(* IEC 61131-3 sources: RL_MAR/experiments/comparison/llm4plc/results/Qwen-Qwen3.5-9B_20260506_150728/20260506_174552, 3 files *)

(* ---- generated_code_iteration_0.st ---- *)
START_ST
FUNCTION_BLOCK SolarPanelTracking
VAR
    PanelAngle : REAL; (* Output for adjusting the solar panel angle *)
    SunriseTime : TIME := T#6H; (* Set the time for sunrise (6:00 AM) *)
    SunsetTime : TIME := T#18H; (* Set the time for sunset (6:00 PM) *)
    NoonTime : TIME := T#12H; (* Set the time for solar noon (12:00 PM) *)
    MorningAngle : REAL := 30.0; (* Set the morning angle for panels *)
    NoonAngle : REAL := 60.0; (* Set the noon angle for panels *)
    EveningAngle : REAL := 30.0; (* Set the evening angle for panels *)
END_VAR
VAR_INPUT
    CurrentTime : TIME;
    SolarIntensity : REAL;
END_VAR
VAR
    state : INT; (* The FSM state variable (0=Night, 1=Morning, 2=Evening, 3=Override) *)
    prevState : INT; (* To track previous state if needed for complex logic *)
    currentAngle : REAL; (* Temporary variable to hold the calculated angle before assignment to output *)
END_VAR

(* Initialize state if this is the first execution or reset logic *)
IF NOT (CurrentTime > T#0) OR (CurrentTime < T#0) THEN
    state := 0;
ELSE
    (* Determine current state based on logic plan *)
    (* STATE 3: HIGH_INTENSITY_OVERRIDE_MODE takes precedence *)
    IF SolarIntensity >= 90.0 THEN
        state := 3;
    (* STATE 0: NIGHT_MODE *)
    ELSIF (CurrentTime < SunriseTime) OR (CurrentTime >= SunsetTime) THEN
        state := 0;
    (* STATE 1: MORNING_MODE *)
    ELSIF CurrentTime < NoonTime THEN
        state := 1;
    (* STATE 2: EVENING_MODE *)
    ELSE
        state := 2;
    END_IF;
END_IF;

(* Assign output based on the determined state *)
CASE state OF
    0: (* NIGHT_MODE *)
        currentAngle := 0.0;
    1: (* MORNING_MODE *)
        currentAngle := MorningAngle;
    2: (* EVENING_MODE *)
        currentAngle := EveningAngle;
    3: (* HIGH_INTENSITY_OVERRIDE_MODE *)
        currentAngle := NoonAngle;
    ELSE
        currentAngle := 0.0; (* Default safety value *)
END_CASE;

(* Update the output variable *)
PanelAngle := currentAngle;

END_FUNCTION_BLOCK
END_ST

(* ---- generated_code_iteration_1.st ---- *)
START_REASON
The validation feedback indicates a CODESYS compiler error: "应该用表达式代替 'T#0'" (Should use an expression instead of 'T#0').

In IEC 61131-3 Structured Text (ST), the literal `T#0` (representing 0 time) is often not accepted directly in boolean comparisons like `CurrentTime > T#0` or `CurrentTime < T#0` because the compiler expects a specific time expression or a comparison against a valid time value that resolves to a boolean context correctly in all dialects.

The standard and most robust way to check if a `TIME` variable is zero is to compare it against `T#0S` (0 seconds) or simply `0` if the context allows, but specifically for `TIME` types, `T#0S` is the explicit zero time duration. However, the most common fix for this specific "expression" error in CODESYS when comparing a TIME variable to zero is to compare it against `T#0S` or to check if the time is less than or equal to `T#0S`.

Another interpretation of the error "use an expression" is that `T#0` might be interpreted as an incomplete time specification in some strict modes, whereas `T#0S` (0 Seconds) is a complete, unambiguous expression.

Additionally, looking at the logic:
`IF NOT (CurrentTime > T#0) OR (CurrentTime < T#0) THEN`
This logic attempts to catch if `CurrentTime` is exactly `T#0`.
If we replace `T#0` with `T#0S`, it becomes a valid time expression.

Let's refine the logic to be safer and strictly compliant:
Instead of `CurrentTime > T#0`, we should use `CurrentTime > T#0S`.
The condition `NOT (CurrentTime > T#0S) OR (CurrentTime < T#0S)` effectively checks if `CurrentTime` is equal to `T#0S`.

Wait, there is a simpler pattern often required by CODESYS for zero checks on TIME:
`CurrentTime <= T#0S` covers 0 and negative times (though TIME is usually unsigned or wraps).
However, the specific error message "use an expression" usually targets the literal `T#0`. Replacing it with `T#0S` is the standard fix.

Let's apply `T#0S` to the comparisons.

Also, I will ensure the variable declarations and structure remain strictly as FUNCTION_BLOCK with correct `END_VAR` usage.

Corrected Logic:
Replace `T#0` with `T#0S`.

START_ST
FUNCTION_BLOCK SolarPanelTracking
VAR
    PanelAngle : REAL; (* Output for adjusting the solar panel angle *)
    SunriseTime : TIME := T#6H; (* Set the time for sunrise (6:00 AM) *)
    SunsetTime : TIME := T#18H; (* Set the time for sunset (6:00 PM) *)
    NoonTime : TIME := T#12H; (* Set the time for solar noon (12:00 PM) *)
    MorningAngle : REAL := 30.0; (* Set the morning angle for panels *)
    NoonAngle : REAL := 60.0; (* Set the noon angle for panels *)
    EveningAngle : REAL := 30.0; (* Set the evening angle for panels *)
END_VAR
VAR_INPUT
    CurrentTime : TIME;
    SolarIntensity : REAL;
END_VAR
VAR
    state : INT; (* The FSM state variable (0=Night, 1=Morning, 2=Evening, 3=Override) *)
    prevState : INT; (* To track previous state if needed for complex logic *)
    currentAngle : REAL; (* Temporary variable to hold the calculated angle before assignment to output *)
END_VAR

(* Initialize state if this is the first execution or reset logic *)
(* Fixed: Replaced T#0 with T#0S to satisfy CODESYS expression requirement *)
IF NOT (CurrentTime > T#0S) OR (CurrentTime < T#0S) THEN
    state := 0;
ELSE
    (* Determine current state based on logic plan *)
    (* STATE 3: HIGH_INTENSITY_OVERRIDE_MODE takes precedence *)
    IF SolarIntensity >= 90.0 THEN
        state := 3;
    (* STATE 0: NIGHT_MODE *)
    ELSIF (CurrentTime < SunriseTime) OR (CurrentTime >= SunsetTime) THEN
        state := 0;
    (* STATE 1: MORNING_MODE *)
    ELSIF CurrentTime < NoonTime THEN
        state := 1;
    (* STATE 2: EVENING_MODE *)
    ELSE
        state := 2;
    END_IF;
END_IF;

(* Assign output based on the determined state *)
CASE state OF
    0: (* NIGHT_MODE *)
        currentAngle := 0.0;
    1: (* MORNING_MODE *)
        currentAngle := MorningAngle;
    2: (* EVENING_MODE *)
        currentAngle := EveningAngle;
    3: (* HIGH_INTENSITY_OVERRIDE_MODE *)
        currentAngle := NoonAngle;
    ELSE
        currentAngle := 0.0; (* Default safety value *)
END_CASE;

(* Update the output variable *)
PanelAngle := currentAngle;

END_FUNCTION_BLOCK
END_ST
END_REASON

(* ---- generated_code_iteration_2.st ---- *)
START_REASON
The previous code failed due to two critical issues:
1.  **Encoding Error**: The error "illegal multibyte sequence" at position 79 indicates that the code contained Chinese characters (likely from the comments explaining the fix). The IEC 61131-3 standard and CODESYS compilers require the source code to be in ASCII or UTF-8. Any non-ASCII characters (like Chinese explanations) will cause a compilation failure. I must remove all Chinese text and replace it with English comments.
2.  **Logic/Expression Error**: The previous attempt to fix `T#0` by using `T#0S` was correct in principle, but the logic `NOT (CurrentTime > T#0S) OR (CurrentTime < T#0S)` is mathematically redundant and potentially confusing. Since `TIME` in PLCs is typically unsigned, `CurrentTime < T#0S` is always false. The condition effectively checks if `CurrentTime == T#0S`. A cleaner, more robust way to handle the "zero time" check or simply ensure the variable is initialized is to compare against `T#0S` directly or ensure the logic flow doesn't rely on ambiguous zero checks unless necessary. However, the primary blocker was the encoding. I will remove the specific `T#0` vs `T#0S` debate and use `T#0S` as the explicit zero time constant, which is the standard fix for the "expression" error, while ensuring all comments are English.

I will now generate the clean, ASCII-compliant, and logically sound Structured Text code.
END_REASON
START_ST
FUNCTION_BLOCK SolarPanelTracking
VAR
    PanelAngle : REAL;
    SunriseTime : TIME := T#6H;
    SunsetTime : TIME := T#18H;
    NoonTime : TIME := T#12H;
    MorningAngle : REAL := 30.0;
    NoonAngle : REAL := 60.0;
    EveningAngle : REAL := 30.0;
END_VAR
VAR_INPUT
    CurrentTime : TIME;
    SolarIntensity : REAL;
END_VAR
VAR
    state : INT;
    currentAngle : REAL;
END_VAR

(* Initialize state: Check if time is zero or invalid *)
IF CurrentTime = T#0S THEN
    state := 0;
ELSE
    (* Determine current state based on logic plan *)
    (* STATE 3: HIGH_INTENSITY_OVERRIDE_MODE takes precedence *)
    IF SolarIntensity >= 90.0 THEN
        state := 3;
    (* STATE 0: NIGHT_MODE *)
    ELSIF (CurrentTime < SunriseTime) OR (CurrentTime >= SunsetTime) THEN
        state := 0;
    (* STATE 1: MORNING_MODE *)
    ELSIF CurrentTime < NoonTime THEN
        state := 1;
    (* STATE 2: EVENING_MODE *)
    ELSE
        state := 2;
    END_IF;
END_IF;

(* Assign output based on the determined state *)
CASE state OF
    0: (* NIGHT_MODE *)
        currentAngle := 0.0;
    1: (* MORNING_MODE *)
        currentAngle := MorningAngle;
    2: (* EVENING_MODE *)
        currentAngle := EveningAngle;
    3: (* HIGH_INTENSITY_OVERRIDE_MODE *)
        currentAngle := NoonAngle;
    ELSE
        currentAngle := 0.0; (* Default safety value *)
END_CASE;

(* Update the output variable *)
PanelAngle := currentAngle;

END_FUNCTION_BLOCK
END_ST
